PROGRAM MAIN
VAR
	basgMotion : MotionControl;
	i: INT;
END_VAR

basgMotion(HMI_MODE:=TRUE);

END_PROGRAM

(* stored: Version 1.1.0.1, ProductVersion 3.1.0.36
   POU MAIN: Id {252640da-6020-4c12-a241-c1e4382f809e}, SpecialFunc None *)
